SUBAPPLICATION Uebung_012f_AR2 (* Numeric Value Input PHYS und Speichern NVS mit Subapp (AR2 Adapter, echter in sich geschlossener Baustein) *)
  (* Standard: 61499-2; Description: Copyright (c) 2026 Meisterschulen am Ostbahnhof This program and the accompanying materials are made available under the terms of the Eclipse Public License 2.0 which is available at https://www.eclipse.org/legal/epl-2.0/ SPDX-License-Identifier: EPL-2.0 *)
  (* Version 1.0, 2026-08-31, Franz Höpfinger, Meisterschulen am Ostbahnhof, AR2 variant of Uebung_012f_AR - NVS_IN_AND_STORE_AR2 (NumericValue_TO_AR2 + NVS_AR2, echt selbstspeichernd) statt NVS_IN_AND_STORE_AR (NumericValue_PHYSA + NVS_AR) *)
  PACKAGE Uebungen;
  IMPORT Uebungen::const::NVS::NVS_Keys::KEY_I1_STORE;
  IMPORT Uebungen::const::UT::DefaultPool_Numeric::InputNumber_I3_N;
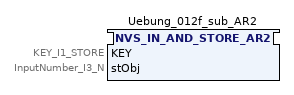
  SUBAPPS
    Uebung_012f_sub_AR2 : MyLib::sys::NVS_IN_AND_STORE_AR2(KEY := KEY_I1_STORE, stObj := InputNumber_I3_N);
  END_SUBAPPS
END_SUBAPPLICATION
